// TIA Portal V20 export
FUNCTION "StepToString" : String   // FC89, SCL
// stored: Namespace Unit1.Em6, SetENOAutomatically false
   VAR_INPUT
      StepDINT : DInt;   // DINT value of the step
   END_VAR
BEGIN
   // Translates shared vision sequence step numbers to step names
   // Sequence-specific duplicate numbers are expressed as combined labels

   CASE #StepDINT OF
       1:
           #StepToString := 'Idle';

       101:
           #StepToString := 'JOB[1] Condition';
       111:
           #StepToString := 'Axis Homed / Controller Ready / QR Ready';
       121:
           #StepToString := 'Axis HomePos Check / Gauge R&R Count Reset';
       131:
           #StepToString := 'Vision Pusher Support WorkPos Check';
       191:
           #StepToString := 'JOB[1] Step End';

       201:
           #StepToString := 'JOB[2] Condition';
       211:
           #StepToString := 'Axis WorkPos / Vision Trigger / QR Trigger';
       291:
           #StepToString := 'JOB[2] Step End';

       301:
           #StepToString := 'JOB[3] Condition';
       311:
           #StepToString := 'Vision Unit AxisZ HomePos Command';
       391:
           #StepToString := 'JOB[3] Step End';

       901:
           #StepToString := 'Immediate Stop';

       1001:
           #StepToString := 'JOB[10] Condition';
       1011:
           #StepToString := 'Vision Unit AxisZ WorkPos Command';
       1021:
           #StepToString := 'Vision Controller Trigger & QR Reader Trigger';
       1031:
           #StepToString := 'Vision Unit AxisZ HomePos Command';
       1091:
           #StepToString := 'JOB[10] Step End';

       9001:
           #StepToString := 'Immediate Stop';

       ELSE
           #StepToString := 'N/A';

   END_CASE;
END_FUNCTION
